// TIA Portal V19 export
FUNCTION_BLOCK "TYPIC_C501_IF_JKP"   // FB35, FBD
TITLE = TYPIC_C501_IF_JKP: Jockeypomp
{ S7_Optimized_Access := 'TRUE' }
AUTHOR : OCOTECH
FAMILY : Typical
NAME : C501.706
// Logisch Object Besturing: C501.706
// 
// De interne functie pomp verzorgt de interne besturing, bewaking en fysieke aansturing van een jockeypomp behorend tot de brandblusinstallatie.
// stored: MemoryReserve 10, SetENOAutomatically false
   VAR_INPUT
      PULS_100ms { ExternalAccessible := 'False'; ExternalVisible := 'False'; ExternalWritable := 'False'} : Bool;   // Puls, 1 PLC-cyclus hoog, 1 keer per 100 ms
      PULS_1s { ExternalAccessible := 'False'; ExternalVisible := 'False'; ExternalWritable := 'False'} : Bool;   // Puls, 1 PLC-cyclus hoog, 1 keer per seconde
      EXT_HW { ExternalAccessible := 'False'; ExternalVisible := 'False'; ExternalWritable := 'False'} : Bool;   // Sturings hardware (PLC) bewaking (1 = OK)
      IN_AAN { ExternalAccessible := 'False'; ExternalVisible := 'False'; ExternalWritable := 'False'} : Bool;   // Terugmelding aansturing
      IN_AUT_C501 { ExternalAccessible := 'False'; ExternalVisible := 'False'; ExternalWritable := 'False'} : Bool;   // Beveiligingen: serie geschakelde terugmelding (1= OK)
      IN_AUT { ExternalAccessible := 'False'; ExternalVisible := 'False'; ExternalWritable := 'False'} : Bool;   // Status thermische beveiliging (1 = OK)
      IN_SCW { ExternalAccessible := 'False'; ExternalVisible := 'False'; ExternalWritable := 'False'} : Bool;   // Werkschakelaar (1 = Aan)
      IN_DME_STO { ExternalAccessible := 'False'; ExternalVisible := 'False'; ExternalWritable := 'False'} : Bool;   // Filterbewaking storing (0 = Storing)
      CFG_TYD_FB { ExternalAccessible := 'False'; ExternalVisible := 'False'; ExternalWritable := 'False'} : Time;   // Vertragingstijd storing foute terugmelding
   END_VAR
   VAR_OUTPUT
      VAR_IF_JKP { ExternalAccessible := 'False'; ExternalVisible := 'False'; ExternalWritable := 'False'} : "C501_VAR_IF_JKP_TYPIC";   // Struct met alle variabelen naar bovenliggende functies
      OUT_AAN { ExternalAccessible := 'False'; ExternalVisible := 'False'; ExternalWritable := 'False'} : Bool;   // Aansturen pomp
   END_VAR
   VAR_IN_OUT
      STU_IF_JKP : "C501_STU_IF_JKP_TYPIC";   // Struct met alle sturingen van de subfunctie (SF) jockeypomp van 3B
   END_VAR
   VAR
      BED : Struct   // Bedieningen
         REM : Bool;   // Bediening om pomp in Remote te schakelen (indien IN_HND = 0)
         FWD : Bool;   // Bediening om pomp in hand te schakelen en te starten
         STOP : Bool;   // Bediening om pomp in hand te schakelen en te stoppen
         RES : Bool;   // Reset storingen
      END_STRUCT;
      STO { ExternalWritable := 'False'} : Struct   // Storingen
         A001 : Bool;   // Beveiliging aangesproken
         A002 : Bool;   // Filter vervuild
         A003 : Bool;   // Storing van de motorbeveiliging van de pomp
         AT01 : Bool;   // Discordantie motor: terugmelding niet ontvangen
         AT02 : Bool;   // Discordantie motor: terugmelding blijft aanwezig
         M001 : Bool;   // Werkschakelaar uitgeschakeld
         M002 : Bool;   // Melding: Pomp heeft te lang niet gedraaid. Periodiek onderhoud nodig
      END_STRUCT;
      VAR { ExternalWritable := 'False'} : Struct   // Variabelen
         STS_AAN : Bool;   // Pomp draait
         BMO_HAND : Bool;   // Pomp in hand geschakeld
         TYD_TOT_AAN { ExternalAccessible := 'False'; ExternalVisible := 'False'} : LInt;   // Totaal aantal draaiuren in seconden
         TYD_TOT_AAN_UUR { ExternalAccessible := 'False'; ExternalVisible := 'False'} : LInt;   // Totaal aantal draaiuren (in uren)
         TYD_AAN { ExternalAccessible := 'False'; ExternalVisible := 'False'} : Int;   // Aantal seconden dat pomp aangeschakeld is
         TYD_UIT { ExternalAccessible := 'False'; ExternalVisible := 'False'} : Int;   // Aantal seconden dat pomp uitgeschakeld is
         EXT_HW { ExternalAccessible := 'False'; ExternalVisible := 'False'} : Bool;   // Sturings hardware (PLC) in storing
      END_STRUCT;
   END_VAR
BEGIN

REGION Network 1: START
END_REGION

REGION Network 2: +++ Storingen +++
   // Verwerken van de storingsmeldingen (inputs).
END_REGION

REGION Network 3: Storing A001: Beveiliging aangesproken
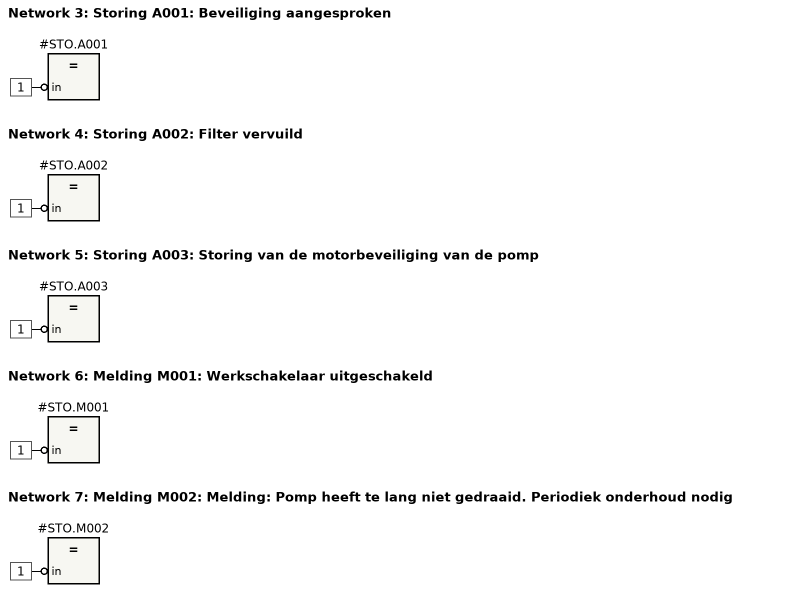
   #STO.A001 := NOT 1;
END_REGION

REGION Network 4: Storing A002: Filter vervuild
   #STO.A002 := NOT 1;
END_REGION

REGION Network 5: Storing A003: Storing van de motorbeveiliging van de pomp
   #STO.A003 := NOT 1;
END_REGION

REGION Network 6: Melding M001: Werkschakelaar uitgeschakeld
   #STO.M001 := NOT 1;
END_REGION

REGION Network 7: Melding M002: Melding: Pomp heeft te lang niet gedraaid. Periodiek onderhoud nodig
   #STO.M002 := NOT 1;
END_REGION

REGION Network 8: +++ Motorsturing +++
   // Aansturen en bewaking van de motor.
END_REGION

REGION Network 9: +++ Urentellers +++
   // Tellen van de tijdsduur dat motor draait of stilstaat.
END_REGION

REGION Network 10 (SCL): EINDE
   // Variabelen van intern scada rakvlak naar outputs copieren
   #VAR_IF_JKP.STS_AAN := #VAR.STS_AAN;
   #VAR_IF_JKP.BMO_HAND := #VAR.BMO_HAND;
   #VAR_IF_JKP.TYD_TOT_AAN := #VAR.TYD_TOT_AAN;
   #VAR_IF_JKP.TYD_TOT_AAN_UUR := #VAR.TYD_TOT_AAN_UUR;
   #VAR_IF_JKP.TYD_AAN := #VAR.TYD_AAN;
   #VAR_IF_JKP.TYD_UIT := #VAR.TYD_UIT;
   #VAR_IF_JKP.EXT_HW := #VAR.EXT_HW;
   #VAR_IF_JKP.STO := #STO;
END_REGION
END_FUNCTION_BLOCK
